PROGRAM MAIN
VAR
  LocalPermit : BOOL;
END_VAR


Plant.PumpAlpha(Start := LocalPermit);
Plant.ValveCommand := LocalPermit;
// Plant.DeprecatedValve := TRUE;

END_PROGRAM
